{attribute 'GeneratedUsingTerminal: EM7004-0000-0017'}
{attribute addProperty BoxType "EM7004-0000-0017"}
{attribute addProperty Id "ControlAT %Q*Control_17BA1FC21"}
{attribute addProperty CRC "2393621028"}
{attribute addProperty Size "1"}
TYPE PLS_Outputs_8EABC224 :
STRUCT
	{attribute addProperty Name "Control"}
	Control AT %Q* : Control_17BA1FC2;
END_STRUCT
END_TYPE

(* stored: Version 1.2.0.0, ProductVersion 3.1.4024.9
   DUT PLS_Outputs_8EABC224: Id {b8be501a-8323-4f5b-990b-cc305bcadf19} *)
